{attribute 'qualified_only'}
VAR_GLOBAL
	Ctrl : ST_Machine_Ctrl;
	Status : ST_Machine_Status;
	ServiceCtrl : ST_Machine_ServiceCtrl;
	ServiceStatus : ST_Machine_ServiceStatus;
	Admin : ST_Machine_Admin;
END_VAR

(* stored: Version 1.1.0.1, ProductVersion 3.1.4026.18
   GVL GVL_Remote: Id {083129a8-4d30-4e4f-87c9-f4c66200117e} *)
